# EPICS autosave request: xx_auto_table_settings.req
$(P)$(T).DESC
$(P)$(T).YANG
$(P)$(T).LX
$(P)$(T).LZ
$(P)$(T).SX
$(P)$(T).SY
$(P)$(T).SZ
$(P)$(T).RX
$(P)$(T).RY
$(P)$(T).RZ
$(P)$(T).LEGU
$(P)$(T).AEGU
$(P)$(T).PREC
$(P)$(T).X0
$(P)$(T).Y0
$(P)$(T).Z0
$(P)$(T).AX0
$(P)$(T).AY0
$(P)$(T).AZ0
$(P)$(T).UHX
$(P)$(T).ULX
$(P)$(T).UHY
$(P)$(T).ULY
$(P)$(T).UHZ
$(P)$(T).ULZ
$(P)$(T).UHAX
$(P)$(T).ULAX
$(P)$(T).UHAY
$(P)$(T).ULAY
$(P)$(T).UHAZ
$(P)$(T).ULAZ
